TEXTLIST ADS_ErrorCodes
  1 = 'Internal error'
  6 = 'target port not found. ADS Server not started '
  7 = 'target machine not found. Missing ADS routes '
  13 = 'Port not connected'
  14 = 'Invalid ADS length'
  15 = 'Invalid ADS Net ID'
  18 = 'Port disabled'
  19 = 'Port already connected'
  24 = 'Invalid ADS port'
  26 = 'TCP send error'
  27 = 'Host unreachable'
  28 = 'Invalid AMS fragment'
  1792 = 'error class <device error> '
  1793 = 'Service is not supported by server   '
  1794 = 'invalid index group  '
  1795 = 'invalid index offset    '
  1796 = 'reading/writing not permitted     '
  1797 = 'parameter size not correct'
  1798 = 'invalid parameter value(s)     '
  1799 = 'device is not in a ready state'
  1800 = 'device is busy '
  1801 = 'invalid context (must be in Windows) '
  1802 = 'out of memory '
  1803 = 'invalid parameter value(s)'
  1804 = 'not found (files, ...) '
  1805 = 'syntax error in command or file   '
  1806 = 'objects do not match '
  1807 = 'object already exists '
  1808 = 'symbol not found '
  1809 = 'symbol version invalid Onlinechange Release handle and get a new one '
  1810 = 'server is in invalid state'
  1811 = 'AdsTransMode not supported '
  1812 = 'Notification handle is invalid Onlinechange Release handle and get a new one '
  1813 = 'Notification client not registered  '
  1814 = 'no more notification handles'
  1815 = 'size for watch too big  '
  1816 = 'device not initialized'
  1817 = 'device has a timeout '
  1818 = 'query interface failed'
  1819 = 'wrong interface required'
  1820 = 'class ID is invalid'
  1821 = 'object ID is invalid'
  1822 = 'request is pending  '
  1823 = 'request is aborted'
  1824 = 'signal warning'
  1825 = 'invalid array index   '
  1826 = 'symbol not active Onlinechange Release handle and get a new one '
  1827 = 'access denied  '
  1828 = 'missing license   Activate license for TwinCAT 3 function '
  1836 = 'exception occured during system start  Check each device transistions'
  1856 = 'Error class client error '
  1857 = 'invalid parameter at service '
  1858 = 'polling list is empty'
  1859 = 'var connection already in use '
  1860 = 'invoke ID in use  '
  1861 = 'timeout elapsed   Check ADS routes of sender and receiver and your  firewall setting'
  1862 = 'error in win32 subsystem'
  1863 = 'Invalid client timeout value '
  1864 = 'ads-port not opened'
  1872 = 'internal error in ads sync'
  1873 = 'hash table overflow '
  1874 = 'key not found in hash'
  1875 = 'no more symbols in cache'
  1876 = 'invalid response received'
  1877 = 'sync port is locked'
  0 = 'no error'
   = 'See ADS returncode at the manual'
   = ''
END_TEXTLIST

(* stored: Version 1.1.0.1, ProductVersion 3.1.4024.12
   TextList ADS_ErrorCodes: Id {7e857c75-1e46-4774-9616-08f027937fe7} *)
